// TIA Portal project "烧嘴控制FB" (V17)

(* hardware
DEVICE "PLC_1"  S7-1200 Station
   slot 0: "Rack_0"  S7-1200 Rack  Rack  V1.0
   slot 1: "PLC_1"  CPU 1214C DC/DC/DC  6ES7 214-1AG40-0XB0  V4.5
*)

// ===== PLC "PLC_1"  CPU 1214C DC/DC/DC =====

VAR_GLOBAL   // PLC tag table "IO变量"
   "3#小火反馈" AT %I0.6 : Bool;
   "3#故障反馈" AT %I0.7 : Bool;
   "3#小火" AT %Q0.6 : Bool;
   "3#复位" AT %Q0.7 : Bool;
   "3#大火" AT %Q1.0 : Bool;
   "烧嘴电源" AT %Q4.6 : Bool;
END_VAR

DATA_BLOCK "信号数据"   // DB1
{ S7_Optimized_Access := 'TRUE' }
VERSION : 0.1
   VAR
      测量值1区 : Real;   // 1区温度测量值 DBD0
      设定值1区 : Real;   // 1区温度设定值 DBD84
   END_VAR
BEGIN
END_DATA_BLOCK

DATA_BLOCK "数字量信号"   // DB2
{ S7_Optimized_Access := 'TRUE' }
VERSION : 0.1
   VAR
      自动3号 : Bool;   // 3号自动模式 DBX0.2
      手动小火3号 : Bool;   // 3号手动小火按钮 DBX1.4
      手动大火3号 : Bool;   // 3号手动大火按钮 DBX2.6
      自动复位失败3号 : Bool;   // 自动复位失败标志 DBX4.0
      烧嘴复位 : Bool;   // 复位清零按钮 DBX5.1
      自动复位关闭 : Bool;   // 手动复位关闭 DBX5.2
      超温标志3区 : Bool;   // 3区超温标志 DBX5.5
   END_VAR
BEGIN
END_DATA_BLOCK

FUNCTION_BLOCK "烧嘴控制"   // FB1, LAD
{ S7_Optimized_Access := 'TRUE' }
VERSION : 0.1
   VAR_INPUT
      测量值 : Real;
      设定值 : Real;
      烧嘴电源 : Bool;
      小火反馈 : Bool;
      故障反馈 : Bool;
      手动复位关闭 : Bool;
      自动 : Bool;
      手动小火 : Bool;
      手动大火 : Bool;
      复位清零 : Bool;
   END_VAR
   VAR_OUTPUT
      小火输出 : Bool;
      大火输出 : Bool;
      复位输出 : Bool;
      自动复位失败 : Bool;
      超温标志 : Bool;
   END_VAR
   VAR
      故障定时器 : IEC_TIMER;
      超温阈值 : Real;
      大火下限 : Real;
      大火上限 : Real;
      复位脉冲存储 : Bool;
      复位失败脉冲存储 : Bool;
   END_VAR
   VAR_TEMP   // added for the SCL form of the ladder/FBD networks
      _w1 : Bool;
      _w2 : Bool;
   END_VAR
BEGIN

REGION Network 1
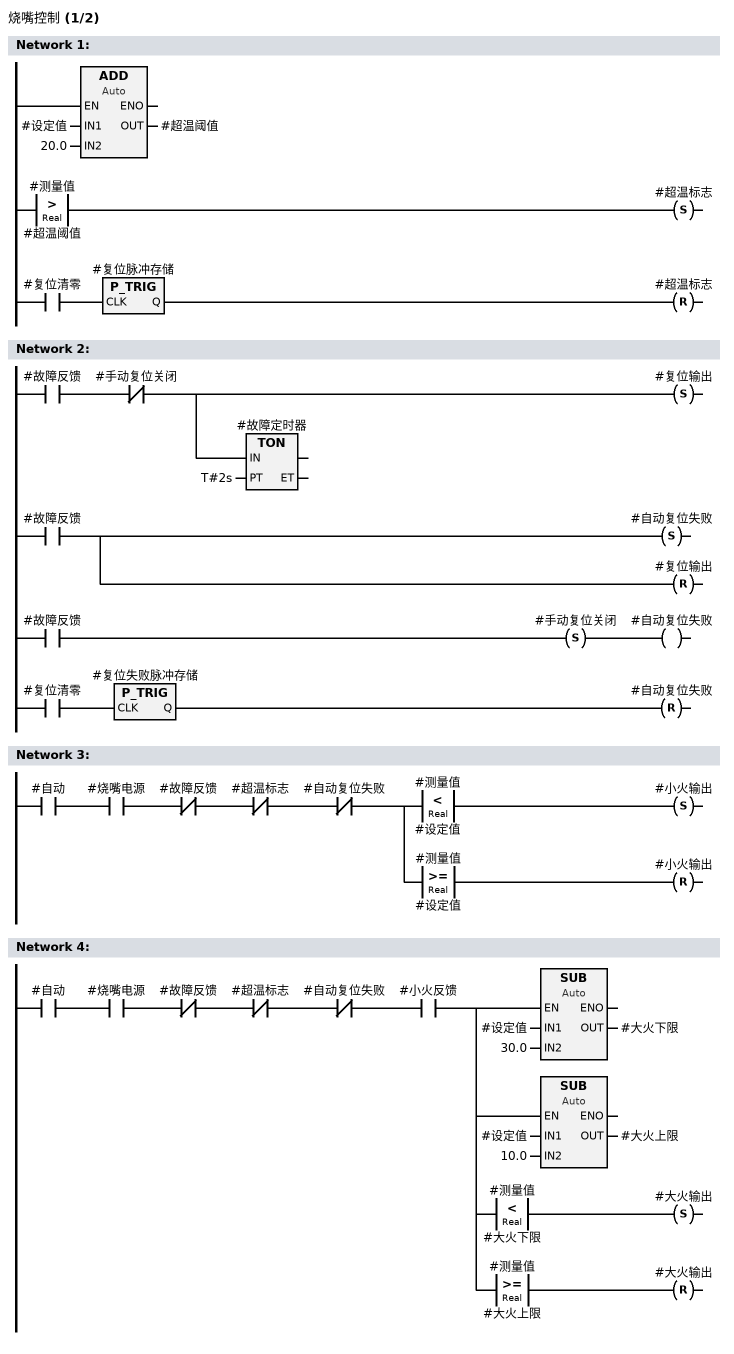
   RUNG wire#powerrail
      { S7_GenerateENO := "TRUE" } Add(in1 := #设定值, in2 := 20.0, out => #超温阈值)
   END_RUNG
   RUNG wire#powerrail
      { S7_Templates := "SrcType := Real" } GT_Contact(in1 := #测量值, in2 := #超温阈值)
      S_Coil( #超温标志 )
   END_RUNG
   RUNG wire#powerrail
      Contact( #复位清零 )
      P_Trig( #复位脉冲存储 )
      R_Coil( #超温标志 )
   END_RUNG
   // the same network as SCL:
   #超温阈值 := #设定值 + 20.0;
   IF #测量值 > #超温阈值 THEN #超温标志 := TRUE; END_IF;
   #_w1 := #复位清零 AND NOT #复位脉冲存储;   // rising edge
   #复位脉冲存储 := #复位清零;
   IF #_w1 THEN #超温标志 := FALSE; END_IF;
END_REGION

REGION Network 2
   #_w1 := #故障反馈 AND NOT #手动复位关闭;
   IF #_w1 THEN #复位输出 := TRUE; END_IF;
   #故障定时器.TON(IN := #_w1, PT := T#2s);
   IF #故障反馈 THEN
       #自动复位失败 := TRUE;
       #复位输出 := FALSE;
       #手动复位关闭 := TRUE;
   END_IF;
   #自动复位失败 := #故障反馈;
   #_w2 := #复位清零 AND NOT #复位失败脉冲存储;   // rising edge
   #复位失败脉冲存储 := #复位清零;
   IF #_w2 THEN #自动复位失败 := FALSE; END_IF;
END_REGION

REGION Network 3
   RUNG wire#powerrail
      Contact( #自动 )
      Contact( #烧嘴电源 )
      I_Contact( #故障反馈 )
      I_Contact( #超温标志 )
      I_Contact( #自动复位失败 )
      wire#w1
      { S7_Templates := "SrcType := Real" } LT_Contact(in1 := #测量值, in2 := #设定值)
      S_Coil( #小火输出 )
   END_RUNG
   RUNG wire#w1
      { S7_Templates := "SrcType := Real" } GE_Contact(in1 := #测量值, in2 := #设定值)
      R_Coil( #小火输出 )
   END_RUNG
   // the same network as SCL:
   #_w1 := #自动 AND #烧嘴电源 AND NOT #故障反馈 AND NOT #超温标志 AND NOT #自动复位失败;
   IF #_w1 AND (#测量值 < #设定值) THEN #小火输出 := TRUE; END_IF;
   IF #_w1 AND (#测量值 >= #设定值) THEN #小火输出 := FALSE; END_IF;
END_REGION

REGION Network 4
   RUNG wire#powerrail
      Contact( #自动 )
      Contact( #烧嘴电源 )
      I_Contact( #故障反馈 )
      I_Contact( #超温标志 )
      I_Contact( #自动复位失败 )
      Contact( #小火反馈 )
      wire#w1
      { S7_GenerateENO := "TRUE" } Sub(in1 := #设定值, in2 := 30.0, out => #大火下限)
   END_RUNG
   RUNG wire#w1
      { S7_GenerateENO := "TRUE" } Sub(in1 := #设定值, in2 := 10.0, out => #大火上限)
   END_RUNG
   RUNG wire#w1
      { S7_Templates := "SrcType := Real" } LT_Contact(in1 := #测量值, in2 := #大火下限)
      S_Coil( #大火输出 )
   END_RUNG
   RUNG wire#w1
      { S7_Templates := "SrcType := Real" } GE_Contact(in1 := #测量值, in2 := #大火上限)
      R_Coil( #大火输出 )
   END_RUNG
   // the same network as SCL:
   #_w1 := #自动 AND #烧嘴电源 AND NOT #故障反馈 AND NOT #超温标志 AND NOT #自动复位失败 AND #小火反馈;
   IF #_w1 THEN
       #大火下限 := #设定值 - 30.0;
       #大火上限 := #设定值 - 10.0;
   END_IF;
   IF #_w1 AND (#测量值 < #大火下限) THEN #大火输出 := TRUE; END_IF;
   IF #_w1 AND (#测量值 >= #大火上限) THEN #大火输出 := FALSE; END_IF;
END_REGION

REGION Network 5
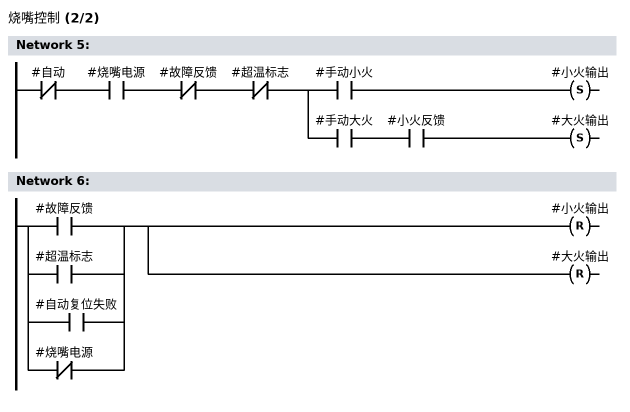
   RUNG wire#powerrail
      I_Contact( #自动 )
      Contact( #烧嘴电源 )
      I_Contact( #故障反馈 )
      I_Contact( #超温标志 )
      wire#w1
      Contact( #手动小火 )
      S_Coil( #小火输出 )
   END_RUNG
   RUNG wire#w1
      Contact( #手动大火 )
      Contact( #小火反馈 )
      S_Coil( #大火输出 )
   END_RUNG
   // the same network as SCL:
   #_w1 := NOT #自动 AND #烧嘴电源 AND NOT #故障反馈 AND NOT #超温标志;
   IF #_w1 AND #手动小火 THEN #小火输出 := TRUE; END_IF;
   IF #_w1 AND #手动大火 AND #小火反馈 THEN #大火输出 := TRUE; END_IF;
END_REGION

REGION Network 6
   RUNG wire#powerrail
      Contact( #故障反馈 )
      wire#w1
      R_Coil( #小火输出 )
   END_RUNG
   RUNG wire#powerrail
      Contact( #超温标志 )
   END_RUNG wire#w1
   RUNG wire#powerrail
      Contact( #自动复位失败 )
   END_RUNG wire#w1
   RUNG wire#powerrail
      I_Contact( #烧嘴电源 )
   END_RUNG wire#w1
   RUNG wire#w1
      R_Coil( #大火输出 )
   END_RUNG
   // the same network as SCL:
   IF #故障反馈 OR #超温标志 OR #自动复位失败 OR NOT #烧嘴电源 THEN
       #小火输出 := FALSE;
       #大火输出 := FALSE;
   END_IF;
END_REGION
END_FUNCTION_BLOCK

ORGANIZATION_BLOCK "Main"   // OB1, SCL, ProgramCycle
{ S7_Optimized_Access := 'TRUE' }
VERSION : 0.1
   VAR_INPUT
      Initial_Call : Bool;   // Initial call of this OB
      Remanence : Bool;   // =True, if remanent data are available
   END_VAR
BEGIN
   "烧嘴控制"(
          测量值      := "信号数据"."测量值1区",
          设定值      := "信号数据"."设定值1区",
          烧嘴电源    := "烧嘴电源",
          小火反馈    := "3#小火反馈",
          故障反馈    := "3#故障反馈",
          手动复位关闭 := "数字量信号"."自动复位关闭",
          自动        := "数字量信号"."自动3号",
          手动小火    := "数字量信号"."手动小火3号",
          手动大火    := "数字量信号"."手动大火3号",
          复位清零    := "数字量信号"."烧嘴复位",
          小火输出    => "3#小火",
          大火输出    => "3#大火",
          复位输出    => "3#复位",
          自动复位失败 => "数字量信号"."自动复位失败3号",
          超温标志    => "数字量信号"."超温标志3区"
   );
END_ORGANIZATION_BLOCK